(* PLC project Unnamed, Unknown Unnamed 1 *)
(* stored: creationDateTime 2021-09-19T16:21:08, modificationDateTime 2021-09-19T17:51:00 *)

PROGRAM program0
  VAR
    LocalVar0 : BOOL;
    LocalVar1 : BOOL;
    LocalVar2 : BOOL;
    LocalVar3 : BOOL;
  END_VAR

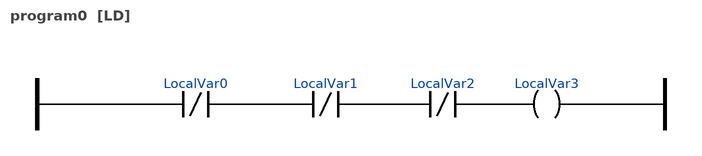
(* LD diagram, written out as Structured Text *)
LocalVar3 := NOT LocalVar0 AND NOT LocalVar1 AND NOT LocalVar2;
END_PROGRAM

CONFIGURATION Config0
  RESOURCE Res0 ON PLC
    TASK task0(INTERVAL := T#20ms, PRIORITY := 0);
    PROGRAM instance0 WITH task0 : program0;
  END_RESOURCE
END_CONFIGURATION
